PROGRAM Systemparameter
VAR
	iState			:eSystemState;
	
	bEinschalten	:BOOL;
	bAusschalten	:BOOL;
	bStarten		:BOOL;
	bStoppen		:BOOL;
	bFehler			:BOOL;
	bResetten		:BOOL;
	bAbgeschlossen	:BOOL;
END_VAR

GVL.SystemState := iState;

CASE iState OF
	0:	// AUS
			// DO
			IF Anlage.UR5.P_State = 1 THEN
				bEinschalten := TRUE;
			END_IF
			
			// TRANSITION
			IF bEinschalten THEN
				bEinschalten := FALSE;
				iState := 1;
			END_IF
		
			
	1:	// BEREIT
			// DO
			IF Anlage.UR5.P_State = 3 THEN
				bStarten := TRUE;
			END_IF
			
			IF Anlage.UR5.P_State = 0 THEN
				bAusschalten := TRUE;
			END_IF
			
			IF GVL.Error THEN
				bFehler := TRUE;
			END_IF
			
			// TRANSITION
			IF bStarten THEN
				bStarten := FALSE;
				iState := 2;
			END_IF
			
			IF bAusschalten THEN
				bAusschalten := FALSE; 
				iState := 0;
			END_IF
			
			IF bFehler THEN
				bFehler := FALSE;
				iState := 4;
			END_IF
			
	2:	// LAUFEND
			// DO
			IF GVL.SystemCommand = 3 THEN
				bStoppen := TRUE;
			END_IF
			
			IF Anlage.UR5.P_State = 1 THEN
				bAbgeschlossen := TRUE;
			END_IF
			
			IF GVL.Error THEN
				bFehler := TRUE;
			END_IF
			
			// TRANSITION
			IF bStoppen THEN
				bStoppen := FALSE;
				iState := 3;
			END_IF
			
			IF bAbgeschlossen THEN
				bAbgeschlossen := FALSE;
				iState := 1;
			END_IF
			
			IF bFehler THEN
				bFehler := FALSE;
				iState := 4;
			END_IF
			
	3:	// GESTOPPT
			// DO
			IF GVL.SystemCommand = 4 THEN
				bResetten := TRUE;
			END_IF
			
			// TRANSITION
			IF bResetten THEN
				bResetten := FALSE;
				iState := 1;
			END_IF
			
	4:	// FEHLER
			// DO
			IF GVL.SystemCommand = 4 THEN
				bResetten := TRUE;
			END_IF
			
			// TRANSITION
			IF bResetten THEN
				bResetten := FALSE;
				iState := 1;
			END_IF
			
END_CASE

END_PROGRAM

(* stored: Version 1.1.0.1
   POU Systemparameter: Id {d1462989-c20e-4f69-a7c2-8b8e9f0c5614}, SpecialFunc None *)
